// TwinCAT 3 PLC project XMLServerTesten
// ProgramVersion: 3.1.4023.0
// libraries:
//   Tc2_Standard, * (Beckhoff Automation GmbH)
//   Tc2_System, * (Beckhoff Automation GmbH)
//   Tc2_Utilities, * (Beckhoff Automation GmbH)
//   Tc2_XmlDataSrv, * (Beckhoff Automation GmbH)
//   Tc3_Module, * (Beckhoff Automation GmbH)
// project tree:
//   DUTs/ Datensatz.TcDUT, XMLHeader.TcDUT (not stored)
//   GVLs/ GVL.TcGVL
//   / PlcTask.TcTTO
//   POUs/ DataLoggingContinue.TcPOU (not stored), fileT_to_sysT.TcPOU (not stored), MAIN.TcPOU (not stored), write_to_Buffer.TcPOU (not stored), write_to_XML_Event.TcPOU (not stored), DataLoggingEvent.TcPOU (not stored), write_to_XML_Continue.TcPOU (not stored)

CONFIGURATION XMLServerTesten
    RESOURCE PLC ON TwinCAT3
        TASK PlcTask(INTERVAL := T#10ms, PRIORITY := 20);
        PROGRAM MAIN WITH PlcTask : MAIN;
    END_RESOURCE
END_CONFIGURATION

// ---- DUTs/Datensatz.TcDUT
TYPE Datensatz :
STRUCT
	Timestamp : STRING ;
	watertemp : LREAL;
	setoutsidetemp : LREAL;
	setwatertemp : LREAL;
	roomtemp1 : LREAL;
	setroomtemp1 : LREAL;
	roomtemp2 : LREAL;
	setroomtemp2 : LREAL;
	a : LREAL;
	b1 : LREAL;
	b2 : LREAL;
END_STRUCT
END_TYPE

// ---- GVLs/GVL.TcGVL
{attribute 'qualified_only'}
VAR_GLOBAL
	
	SetAussenTemp AT %Q*: LREAL := 17;
	SetWasserTemp AT %Q*: LREAL := 90;
	SetRaumTemp1 AT %Q*: LREAL := 20;
	Traum1 AT %I*: LREAL;
	TWasser AT %I*: LREAL;
	Traum2 AT %I*: LREAL;
	setAussenT AT %I*: LREAL;
	setWasserT AT %I*: LREAL;
	a AT %I*: LREAL;
	b1 AT %I*: LREAL;
	b2 AT %I*: LREAL;
	setRaumT1 AT %I*: LREAL;
	setRaumT2 AT %I*: LREAL;
	SetRaumTemp2 AT %Q*: LREAL := 25;
END_VAR
